VAR_GLOBAL CONSTANT
	UNIT_mm : STRING := 'mm';
	UNIT_degree : STRING := 'deg';
	UNIT_radians : STRING := 'rad';
END_VAR

(* stored: Version 1.1.0.1, ProductVersion 3.1.4024.11
   GVL GVL_UnitStrings: Id {b941d280-eea1-4685-b21f-5e664ab0285f} *)
